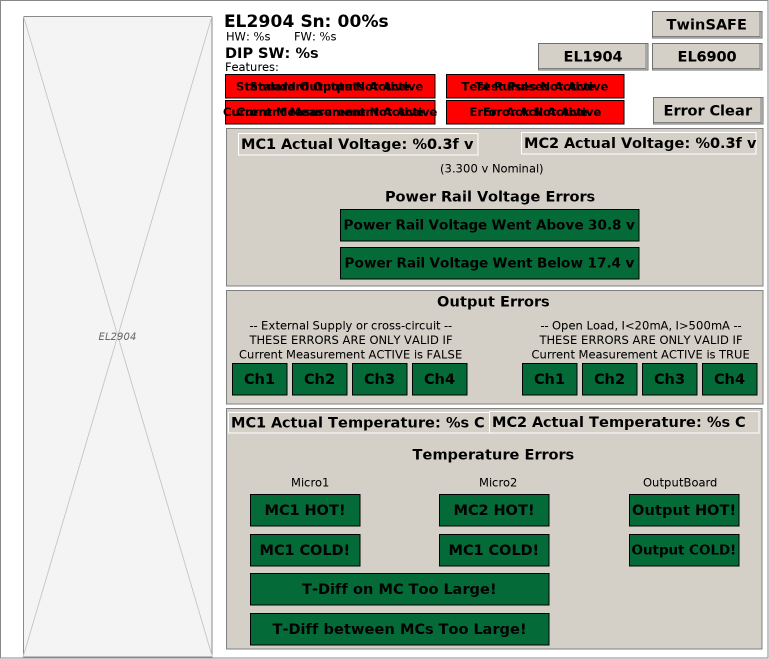
VISUALIZATION EL2904_Specific_Diagnostics  // 769x659
    Button (652,11 110x27), "TwinSAFE"
        OnMouseClick: change screen: TwinSAFE
    Button (652,43 110x27), "EL6900"
        OnMouseClick: change screen: EL6900_Specific_Diagnostics
    Button (538,43 110x27), "EL1904"
        OnMouseClick: change screen: EL1904_Specific_Diagnostics
    Image (23,16 189x641), image: EL2904
    Rectangle (221,10 275x22), "EL2904 Sn: 00%s", text variable: g_dwHMI_EL2904Sn
    Rectangle (223,28 65x17), "HW: %s", text variable: g_sHMI_EL2904_HWvers
    Rectangle (291,28 65x17), "FW: %s", text variable: g_sHMI_EL2904_FWvers
    Rectangle (222,45 164x16), "DIP SW: %s", text variable: g_wHMI_EL2904DSw
    Label (222,59 88x16), "Features:"
    Button (653,97 110x27), "Error Clear"
        OnMouseUp: execute { g_xHMI_EL2904_ErrClearPB := FALSE ; }
        OnMouseDown: execute { g_xHMI_EL2904_ErrClearPB := TRUE ; }
    Rectangle (226,128 537x158)
    Label (433,161 118x15), "(3.300 v Nominal)"
    Rectangle (238,133 240x22), "MC1 Actual Voltage: %0.3f v", text variable: g_wHMI_EL2904PriMC_Volts
    Rectangle (521,132 235x22), "MC2 Actual Voltage: %0.3f v", text variable: g_wHMI_EL2904SecMC_Volts
    Rectangle (226,290 537x114)
    Rectangle (226,408 536x241)
    Rectangle (228,412 264x21), "MC1 Actual Temperature: %s C", text variable: g_wHMI_EL2904PriMCTemp
    Rectangle (489,411 270x22), "MC2 Actual Temperature: %s C", text variable: g_wHMI_EL2904SecMCTemp
    Label (280,474 61x17), "Micro1"
    Label (402,440 183x29), "Temperature Errors"
    Label (225,311 252x58), "-- External Supply or cross-circuit -- THESE ERRORS ARE ONLY VALID IF Current Measurement ACTIVE is FALSE"
    Label (376,185 228x23), "Power Rail Voltage Errors"
    Label (429,287 129x29), "Output Errors"
    Rectangle (340,209 299x32), "Power Rail Voltage Went Above 30.8 v", colour toggle: g_xHMI_EL2904_PwrRailVoltageHi
    Rectangle (340,247 299x32), "Power Rail Voltage Went Below 17.4 v", colour toggle: g_xHMI_EL2904_PwrRailVoltageLo
    Label (515,311 252x58), "-- Open Load, I<20mA, I>500mA -- THESE ERRORS ARE ONLY VALID IF Current Measurement ACTIVE is TRUE"
    Rectangle (232,363 55x32), "Ch1", colour toggle: g_xHMI_EL2904_ExtSup_CrossCirErr_Out1
    Rectangle (292,363 55x32), "Ch2", colour toggle: g_xHMI_EL2904_ExtSup_CrossCirErr_Out2
    Rectangle (352,363 55x32), "Ch3", colour toggle: g_xHMI_EL2904_ExtSup_CrossCirErr_Out3
    Rectangle (412,363 55x32), "Ch4", colour toggle: g_xHMI_EL2904_ExtSup_CrossCirErr_Out4
    Rectangle (522,363 55x32), "Ch1", colour toggle: g_xHMI_EL2904_OutLoadErr_Out1
    Rectangle (582,363 55x32), "Ch2", colour toggle: g_xHMI_EL2904_OutLoadErr_Out2
    Rectangle (642,363 55x32), "Ch3", colour toggle: g_xHMI_EL2904_OutLoadErr_Out3
    Rectangle (702,363 55x32), "Ch4", colour toggle: g_xHMI_EL2904_OutLoadErr_Out4
    Label (468,474 61x17), "Micro2"
    Label (633,474 95x17), "OutputBoard"
    Rectangle (250,494 110x32), "MC1 HOT!", colour toggle: g_xHMI_EL2904_TempErr_OTMc1
    Rectangle (250,534 110x32), "MC1 COLD!", colour toggle: g_xHMI_EL2904_TempErr_UTMc1
    Rectangle (439,494 110x32), "MC2 HOT!", colour toggle: g_xHMI_EL2904_TempErr_OTMc2
    Rectangle (439,534 110x32), "MC1 COLD!", colour toggle: g_xHMI_EL2904_TempErr_UTMc2
    Rectangle (629,494 110x32), "Output HOT!", colour toggle: g_xHMI_EL2904_TempErr_OTOutBoard
    Rectangle (629,534 110x32), "Output COLD!", colour toggle: g_xHMI_EL2904_TempErr_UTOutBoard
    Rectangle (250,573 299x32), "T-Diff on MC Too Large!", colour toggle: g_xHMI_EL2904_TempErr_DiffOnBoard
    Rectangle (250,613 299x32), "T-Diff between MCs Too Large!", colour toggle: g_xHMI_EL2904_TempErr_DiffBetweenMc1Mc2
    Rectangle (225,74 210x24), colour toggle: g_xHMI_EL2904_StandardOuts
    Rectangle (446,74 178x24), colour toggle: g_xHMI_EL2904_TestPulses
    Rectangle (225,100 210x24), colour toggle: g_xHMI_EL2904_CurrentMeas
    Rectangle (446,100 178x24), colour toggle: g_xHMI_EL2904_ErrAck
    Group (241,75 178x23)
        Label (0,0 178x23), "Standard Outputs Not Active", invisible if: g_xHMI_EL2904_StandardOuts
        Label (0,0 178x23), "Standard Outputs Active", invisible if: not g_xHMI_EL2904_StandardOuts
    Group (446,75 178x23)
        Label (0,0 178x23), "Test Pulses Not Active", invisible if: g_xHMI_EL2904_TestPulses
        Label (0,0 178x23), "Test Pulses Active", invisible if: not g_xHMI_EL2904_TestPulses
    Group (226,97 209x30)
        Label (0,0 209x30), "Current Measurement Not Active", invisible if: g_xHMI_EL2904_CurrentMeas
        Label (6,0 197x30), "Current Measurement Active", invisible if: not g_xHMI_EL2904_CurrentMeas
    Group (462,97 147x30)
        Label (0,0 147x30), "Error Ack Not Active", invisible if: g_xHMI_EL2904_ErrAck
        Label (0,0 147x30), "Error Ack Active", invisible if: not g_xHMI_EL2904_ErrAck
END_VISUALIZATION

(* stored: Version 1.1.0.1, ProductVersion 3.1.0.18
   Visu EL2904_Specific_Diagnostics: Id {40e77353-2d0e-4d9d-92e0-7953e3672395} *)
